TEXTLIST AxesMoveVelocityUnitsTextList
  0 = 'degree / s'
  1 = 'arcsec / s'
  2 = 'rad / s'
  3 = 'arcsec / min'
  4 = 'arcsec / hour'
   = ''
END_TEXTLIST

(* stored: Version 1.1.0.1, ProductVersion 3.1.4019.2
   TextList AxesMoveVelocityUnitsTextList: Id {8539a74d-d72e-4ab6-9064-2fd2f0443602} *)
